// SIMATIC S7-200 project (STEP 7-Micro/WIN), CPU 224XP REL 02.01

ORGANIZATION_BLOCK 主程序:OB1
TITLE=程序注释/首次扫描时执行PID子程序
BEGIN
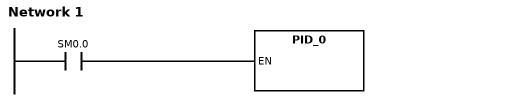
Network 1
LD     SM0.0
CALL   PID_0:SBR0
END_ORGANIZATION_BLOCK

SUBROUTINE_BLOCK PID_0:SBR0
TITLE=程序注释
BEGIN
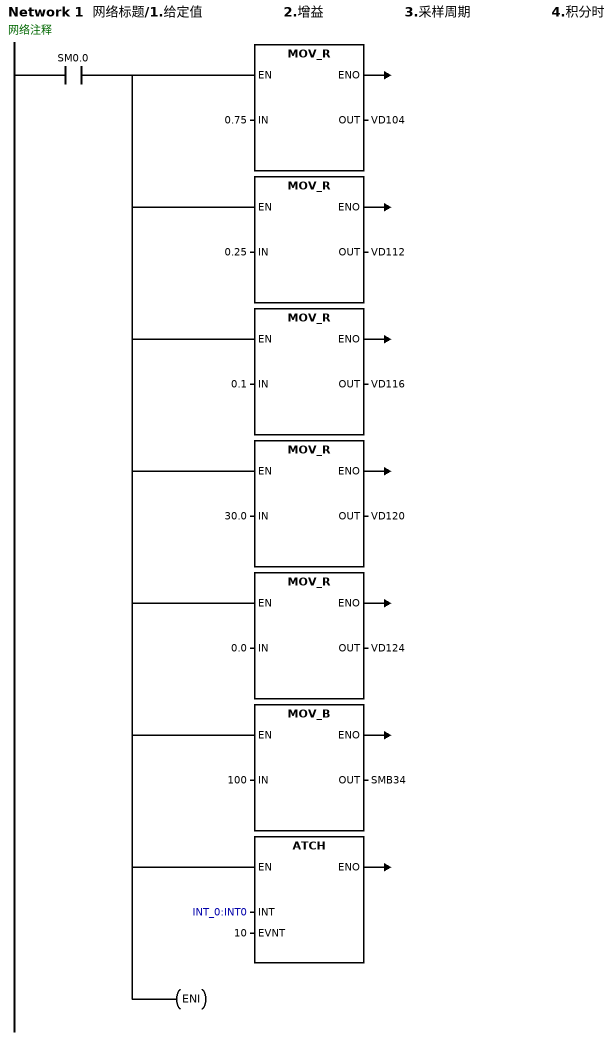
Network 1 // 网络标题/1.给定值
                 2.增益
                 3.采样周期
                 4.积分时间
                 5.微分时间
                 6.100ms定时中断
// 网络注释
LD     SM0.0
MOVR   0.75, VD104
MOVR   0.25, VD112
MOVR   0.1, VD116
MOVR   30.0, VD120
MOVR   0.0, VD124
MOVB   100, SMB34
ATCH   INT_0:INT0, 10
ENI
Network 26 // 网络标题
// 网络注释
END_SUBROUTINE_BLOCK

// SBR1: protected block, not included

INTERRUPT_BLOCK INT_0:INT0
TITLE=中断程序注释
BEGIN
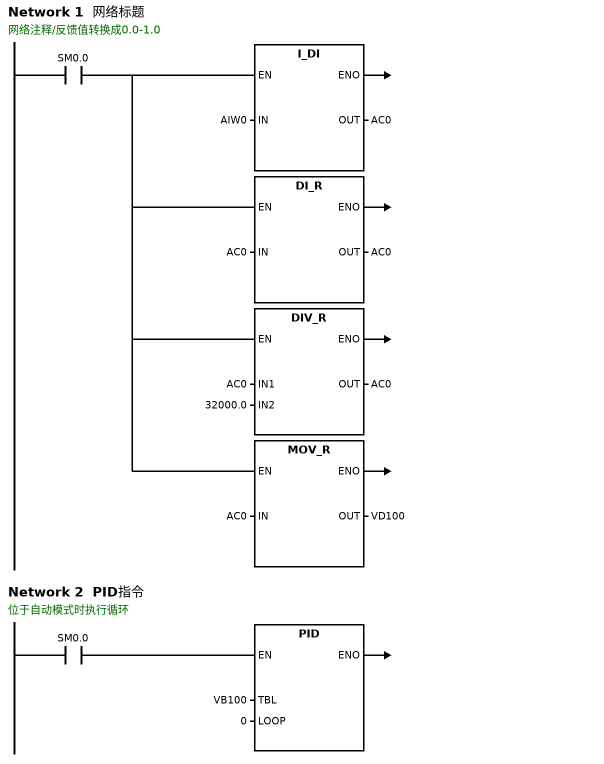
Network 1 // 网络标题
// 网络注释/反馈值转换成0.0-1.0
LD     SM0.0
ITD    AIW0, AC0
DTR    AC0, AC0
/R     32000.0, AC0
MOVR   AC0, VD100
Network 2 // PID指令
// 位于自动模式时执行循环
LD     SM0.0
PID    VB100, 0
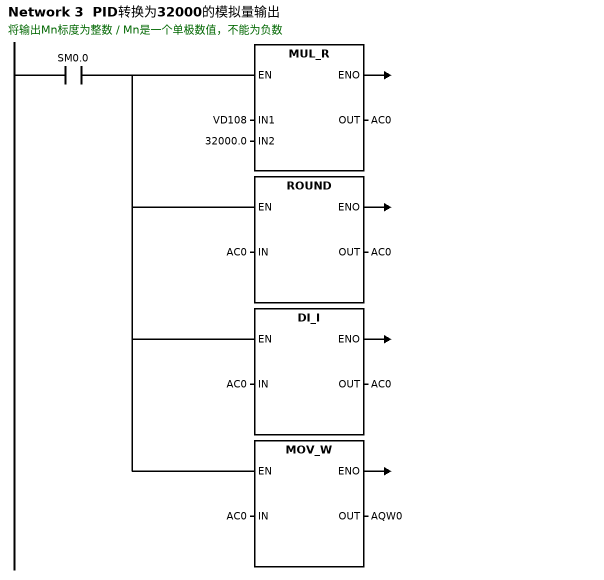
Network 3 // PID转换为32000的模拟量输出
// 将输出Mn标度为整数
// Mn是一个单极数值，不能为负数
LD     SM0.0
MOVR   VD108, AC0
*R     32000.0, AC0
ROUND  AC0, AC0
DTI    AC0, AC0
MOVW   AC0, AQW0
END_INTERRUPT_BLOCK

// INT1: protected block, not included

// (further data pages could not be read)
